FUNCTION_BLOCK STATION3_INFO
  {SET_ATTRIBUTE(OpcUa, SERVICE)}
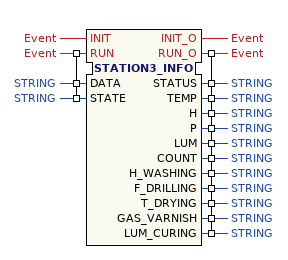
  EVENT_INPUT
    INIT;
    RUN WITH DATA, STATE; {SET_ATTRIBUTE(OpcUa, Method)}
  END_EVENT
  EVENT_OUTPUT
    INIT_O;
    RUN_O WITH STATUS, TEMP, H, P, LUM, COUNT, H_WASHING, F_DRILLING, T_DRYING, GAS_VARNISH, LUM_CURING;
  END_EVENT
  VAR_INPUT
    DATA : STRING;
    STATE : STRING;
  END_VAR
  VAR_OUTPUT
    STATUS : STRING;
    TEMP : STRING;
    H : STRING;
    P : STRING;
    LUM : STRING;
    COUNT : STRING;
    H_WASHING : STRING;
    F_DRILLING : STRING;
    T_DRYING : STRING;
    GAS_VARNISH : STRING;
    LUM_CURING : STRING;
  END_VAR
END_FUNCTION_BLOCK
